GLOBALCONSTANTS DefaultPool_TECU (* Global constants *)
  PACKAGE Uebungen::const::UT::TECU;
  VAR_GLOBAL CONSTANT
    ISO_DESIGNATOR_WIDTH : UINT := 80;
    ISO_DESIGNATOR_HEIGHT : UINT := 80;
    ISO_MASK_SIZE : UINT := 480;
    ISO_VERSION_LABEL : STRING;
    MASK_WIDTH : UINT := 480;
    MASK_HEIGHT : UINT := 480;
    WorkingSet : UINT := 0;
    DataMask_M1 : UINT := 1000;
    Container_Wheel_based_machine_speed : UINT := 3000;
    Container_Ground_based_machine_speed : UINT := 3001;
    Container_Wheel_based_machine_distance : UINT := 3002;
    Container_Rear_PTO_output_shaft_speed : UINT := 3003;
    SoftKeyMask_S1 : UINT := 4000;
    OutputString_km_h : UINT := 11000;
    OutputString_m_s : UINT := 11001;
    OutputString_km : UINT := 11002;
    OutputString_m : UINT := 11003;
    OutputString_1_min : UINT := 11004;
    OutputNumber_Wheel_based_machine_speed_km_h : UINT := 12000;
    OutputNumber_Wheel_based_machine_speed_m_s : UINT := 12001;
    OutputNumber_Ground_based_machine_speed_km_h : UINT := 12002;
    OutputNumber_Ground_based_machine_speed_m_s : UINT := 12003;
    OutputNumber_Wheel_based_machine_distance_km : UINT := 12004;
    OutputNumber_Wheel_based_machine_distance_m : UINT := 12005;
    OutputNumber_Rear_PTO_output_shaft_speed : UINT := 12006;
    Line : UINT := 13000;
    Tractor_wheel_slip : UINT := 20000;
    Battery_disconnect : UINT := 20001;
    Work_distance_travelled : UINT := 20002;
    Tractor_ground_speed : UINT := 20003;
    PTO_output_shaft_speed : UINT := 20004;
    NumberVariable_Wheel_based_machine_speed : UINT := 21000;
    NumberVariable_Ground_based_machine_speed : UINT := 21001;
    NumberVariable_Wheel_based_machine_distance : UINT := 21002;
    NumberVariable_Rear_PTO_output_shaft_speed : UINT := 21003;
    NumberVariable_TECU_Speed_WBSD : UINT := 21024;
    NumberVariable_TECU_Speed_GBSD : UINT := 21025;
    NumberVariable_TECU_Speed_MSS : UINT := 21026;
    NumberVariable_TECU_Speed_VDS : UINT := 21027;
    NumberVariable_TECU_Speed_COGSOG : UINT := 21028;
    NumberVariable_TECU_FHS_Position : UINT := 21029;
    NumberVariable_TECU_RHS_Position : UINT := 21030;
    NumberVariable_TECU_FHS_Force : UINT := 21031;
    NumberVariable_TECU_RHS_Force : UINT := 21032;
    NumberVariable_TECU_FHS_Draft : UINT := 21033;
    NumberVariable_TECU_RHS_Draft : UINT := 21034;
    NumberVariable_TECU_FPTO_Speed : UINT := 21035;
    NumberVariable_TECU_RPTO_Speed : UINT := 21036;
    NumberVariable_TECU_FPTO_SpeedSet : UINT := 21037;
    NumberVariable_TECU_RPTO_SpeedSet : UINT := 21038;
    FontAttributes_OutputNumber : UINT := 23000;
    FontAttributes_OutputString : UINT := 23001;
    LineAttributes : UINT := 24000;
  END_VAR
END_GLOBALCONSTANTS
